(* CODESYS project Buffer Station - Kaid v6.0.project

Project tree, tasks and I/O mapping:
  Device : CODESYS Control Win V3, 3S - Smart Software Solutions GmbH, order no. 305021, version 3.5.11.30
    application Application
      libraries: Standard, * (System); CmpApp, 3.5.11.0 (System)
      task MainTask (cyclic, interval t#20ms, priority 1) calls PLC_PRG
      program PLC_PRG [LD]: A_Reset_Geral
      Symbols
*)

// Device/Application/PLC_PRG
PROGRAM PLC_PRG
VAR
	// Entradas e Controle
	firstScan		: BOOL;
	aux1: BOOL;
	Remover_Plastico	: BOOL := TRUE;
	Remover_Metal		: BOOL := TRUE;
	xStart_Button            : BOOL;
	S_Capacitivo        : BOOL;
	S_Indutivo          : BOOL;
	xReset_Button       : BOOL;
	xStop_Button        : BOOL;

	// Lugares da Rede de Petri (BOOL para Metodologia de Kaid)
	M_P0_Home            : BOOL;
	M_P1_Alimentacao     : BOOL;
	M_P2_Metal           : BOOL;
	M_P2_Plastico        : BOOL;
	M_P3_Desvia_Plastico : BOOL;

	// Sinais de Transição e Flags
	S_T3_Plastico_Out  : BOOL;
	S_T4_Metal_Out : BOOL;
	

	// Atuadores
	Emitter        : BOOL;
	Pusher         : BOOL;
	Conveyor_Motor : INT; // Mantido como INT conforme sua solicitação

	// Temporizadores e Triggers
	T2_Wait_Pos    : TIME := T#2.5S;
	tonPos         : TON;
	trigReset      : R_TRIG;
	
	// Memórias das transições
	M_T0_Start: BOOL;
	M_T1_Metal: BOOL;
	M_T1_Plastico: BOOL;
	M_T2_Wait_Pos: BOOL;
	M_T3_Pla_Out: BOOL;
	M_T4_Metal_Out: BOOL;

END_VAR
VAR // added by the converter: edge detectors and wires of the graphical bodies
    _ft1 : F_TRIG;
END_VAR

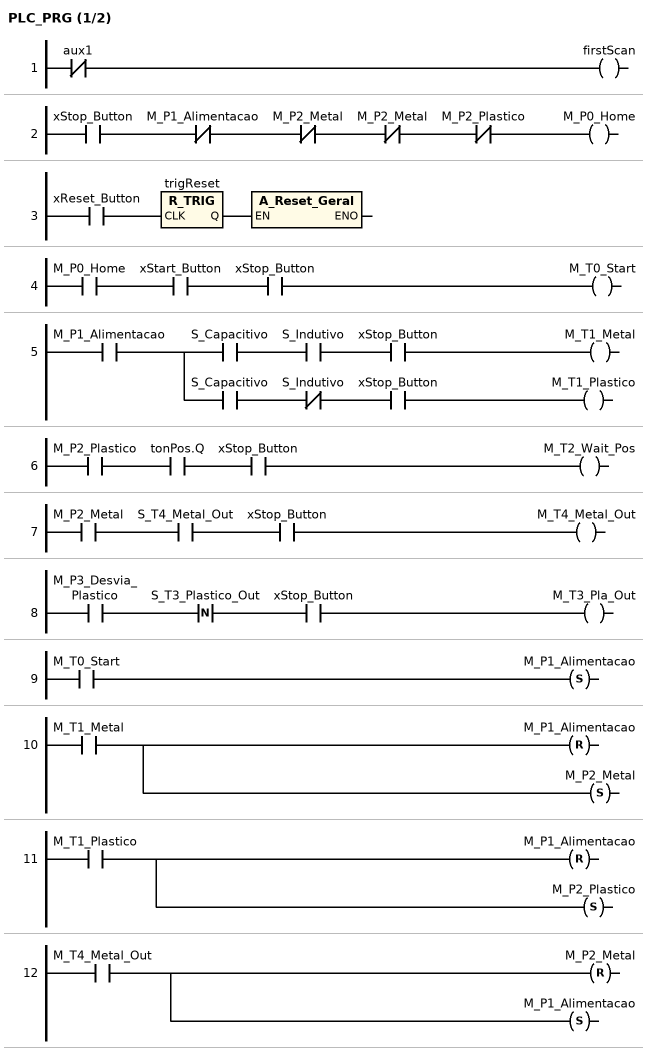
// NETWORK 1
firstScan := NOT aux1;

// NETWORK 2
M_P0_Home := xStop_Button AND NOT M_P1_Alimentacao AND NOT M_P2_Metal AND NOT M_P2_Metal AND NOT M_P2_Plastico;

// NETWORK 3
trigReset(CLK := xReset_Button); // R_TRIG
IF trigReset.Q THEN A_Reset_Geral(); END_IF

// NETWORK 4
M_T0_Start := M_P0_Home AND xStart_Button AND xStop_Button;

// NETWORK 5
M_T1_Metal := M_P1_Alimentacao AND S_Capacitivo AND S_Indutivo AND xStop_Button;
M_T1_Plastico := M_P1_Alimentacao AND S_Capacitivo AND NOT S_Indutivo AND xStop_Button;

// NETWORK 6
M_T2_Wait_Pos := M_P2_Plastico AND tonPos.Q AND xStop_Button;

// NETWORK 7
M_T4_Metal_Out := M_P2_Metal AND S_T4_Metal_Out AND xStop_Button;

// NETWORK 8
_ft1(CLK := S_T3_Plastico_Out);
M_T3_Pla_Out := M_P3_Desvia_Plastico AND _ft1.Q AND xStop_Button;

// NETWORK 9
M_P1_Alimentacao S= M_T0_Start;

// NETWORK 10
M_P1_Alimentacao R= M_T1_Metal;
M_P2_Metal S= M_T1_Metal;

// NETWORK 11
M_P1_Alimentacao R= M_T1_Plastico;
M_P2_Plastico S= M_T1_Plastico;

// NETWORK 12
M_P2_Metal R= M_T4_Metal_Out;
M_P1_Alimentacao S= M_T4_Metal_Out;

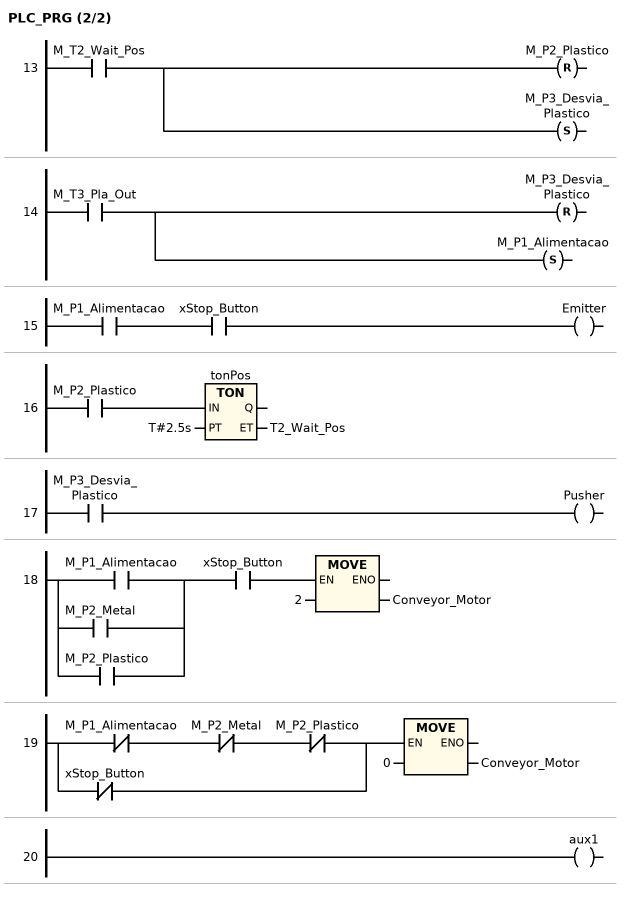
// NETWORK 13
M_P2_Plastico R= M_T2_Wait_Pos;
M_P3_Desvia_Plastico S= M_T2_Wait_Pos;

// NETWORK 14
M_P3_Desvia_Plastico R= M_T3_Pla_Out;
M_P1_Alimentacao S= M_T3_Pla_Out;

// NETWORK 15
Emitter := M_P1_Alimentacao AND xStop_Button;

// NETWORK 16
tonPos(IN := M_P2_Plastico, PT := T#2.5s, ET => T2_Wait_Pos); // TON

// NETWORK 17
Pusher := M_P3_Desvia_Plastico;

// NETWORK 18
IF (M_P1_Alimentacao OR M_P2_Metal OR M_P2_Plastico) AND xStop_Button THEN Conveyor_Motor := 2; END_IF

// NETWORK 19
IF NOT M_P1_Alimentacao AND NOT M_P2_Metal AND NOT M_P2_Plastico OR NOT xStop_Button THEN
    Conveyor_Motor := 0;
END_IF

// NETWORK 20
aux1 := TRUE;

ACTION A_Reset_Geral:
// --- ESTADO INICIAL E CONTROLE ---
aux1   := TRUE;   // O sistema inicia habilitado
Remover_Plastico := TRUE;   // Reset das condições de operação
Remover_Metal    := TRUE;   //
xStart_Button           := FALSE;  // Limpa o comando de partida

// --- LUGARES DA REDE DE PETRI (MARCAÇÃO INICIAL) ---
M_P0_Home            := FALSE;  // Único lugar que inicia com o token
M_P1_Alimentacao     := FALSE;
M_P2_Metal           := FALSE;
M_P2_Plastico        := FALSE;
M_P3_Desvia_Plastico := FALSE;

// --- SINAIS DE TRANSIÇÃO E FLAGS ---
S_T4_Metal_Out := FALSE; // Limpa as memórias de transição
S_T3_Plastico_Out  := FALSE; //

// --- ATUADORES E SAÍDAS ---
Emitter        := FALSE; // Para a geração de novas peças
Pusher         := FALSE; // Recolhe o atuador pneumático
Conveyor_Motor := 0;     // Garante motor parado (Tipo INT)

// --- TEMPORIZADORES E TRIGGERS ---
tonPos(IN := FALSE);     // Reseta o tempo acumulado do timer
trigReset(CLK := FALSE); // Prepara o detector de borda para um novo ciclo
END_ACTION

END_PROGRAM
